PROGRAM P_Demo_F_GetWeekOfTheYear
VAR
    dtProduction  : DATE_AND_TIME := DT#2026-05-11-08:00:00; // 投产日期
    wCalendarWeek : WORD; // ISO 8601 周编号（1~53）
    bRunOnce      : BOOL; // 脉冲触发
END_VAR

// =============================================================================
// 场景：与 MES 系统对接，按 ISO 周编号下发周生产计划「CW19 投产 A 型号」
//
// 价值：1 行得到 ISO 周编号，自动处理跨年情形（12/29 可能属于下年第 1 周）
//
// 验证步骤：
//   1. 引用 Tc2_Utilities
//   2. 编译 + 登录 + 运行
//   3. 强制 bRunOnce := TRUE
//   4. 在线观察 wCalendarWeek = 20（2026-05-11 是 CW20）
//   5. dtProduction := DT#2027-01-01 → wCalendarWeek = 53（属于 2026 第 53 周，跨年规则）
// =============================================================================
wCalendarWeek := F_GetWeekOfTheYear(dtProduction);

END_PROGRAM

(* stored: Version 1.1.0.1, ProductVersion 3.1.4024.5
   POU P_Demo_F_GetWeekOfTheYear: Id {394f83fd-c1d0-59fe-b5a6-f3b706948592}, SpecialFunc None *)
